Yaskawa INFORM job: kufsa_new.JBI

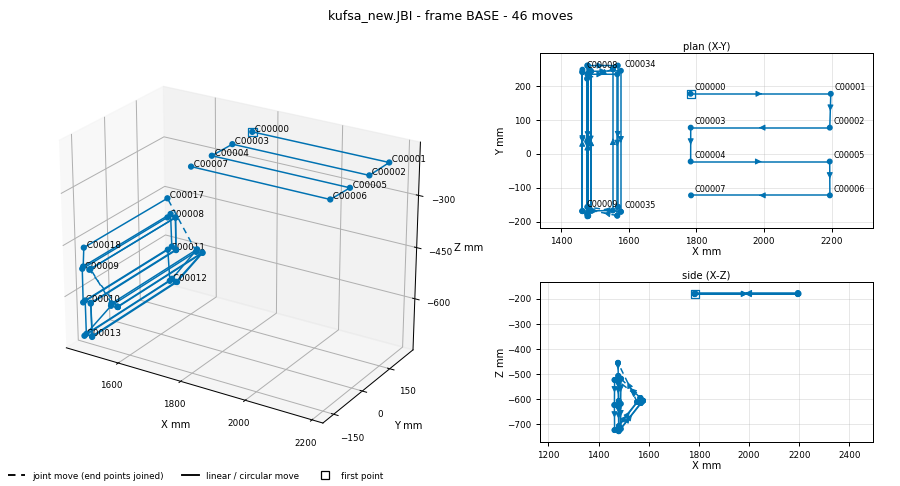
[picture p0: tool path of kufsa_new.JBI in frame BASE, 46 of 52 moves have a stored position in this frame; points joined in program order, loops and branches not executed]
/JOB
//NAME kufsa_new
//POS
///NPOS 46,0,46,0,0,0
///TOOL 0
///POSTYPE BASE
///RECTAN
///RCONF 1,0,0,0,0,0,0,0,0,0,0,0,0,0,0,0,0,0,0,0,0,0,0,0
C00000=1783.333,177.683,-178.952,175.0000,5.0000,90.0000
C00001=2197.437,177.683,-178.952,175.0000,5.0000,90.0000
C00002=2194.402,77.683,-180.929,175.0000,5.0000,90.0000
C00003=1783.689,77.683,-180.929,175.0000,5.0000,90.0000
C00004=1783.507,-22.316,-180.005,175.0000,5.0000,90.0000
C00005=2194.164,-22.316,-180.005,175.0000,5.0000,90.0000
C00006=2194.697,-122.316,-175.996,175.0000,5.0000,90.0000
C00007=1784.686,-122.316,-175.996,175.0000,5.0000,90.0000
C00008=1464.014,241.444,-522.722,175.0000,-89.9999,5.0000
C00009=1464.014,-169.159,-522.722,175.0000,-89.9999,5.0000
C00010=1463.152,-168.687,-622.722,175.0000,-89.9999,5.0000
C00011=1463.152,242.022,-622.722,175.0000,-89.9999,5.0000
C00012=1463.935,248.955,-722.722,175.0000,-89.9999,5.0000
C00013=1463.935,-168.695,-722.722,175.0000,-89.9999,5.0000
C00014=1553.861,-166.978,-610.590,180.0000,-45.0000,0.0000
C00015=1553.861,250.441,-610.590,180.0000,-45.0000,0.0000
C00016=1553.861,250.441,-610.590,180.0000,-45.0000,0.0000
C00017=1477.531,222.423,-454.518,175.0000,-89.9999,5.0000
C00018=1477.531,-177.571,-454.518,175.0000,-89.9999,5.0000
C00019=1478.554,-184.306,-506.723,175.0000,-89.9999,5.0000
C00020=1478.554,235.762,-506.723,175.0000,-89.9999,5.0000
C00021=1480.684,236.380,-606.723,175.0000,-89.9999,5.0000
C00022=1480.684,-183.074,-606.723,175.0000,-89.9999,5.0000
C00023=1480.955,-182.919,-706.723,175.0000,-89.9999,5.0000
C00024=1480.955,235.380,-706.723,175.0000,-89.9999,5.0000
C00025=1566.683,235.369,-594.591,180.0000,-45.0000,0.0000
C00026=1566.683,-182.153,-594.591,180.0000,-45.0000,0.0000
C00027=1566.683,-182.153,-594.591,180.0000,-45.0000,0.0000
C00028=1489.401,-166.687,-517.941,175.0000,-89.9999,5.0000
C00029=1489.401,243.705,-517.941,175.0000,-89.9999,5.0000
C00030=1488.117,245.937,-617.941,175.0000,-89.9999,5.0000
C00031=1488.117,-168.048,-617.941,175.0000,-89.9999,5.0000
C00032=1488.292,-166.510,-717.941,175.0000,-89.9999,5.0000
C00033=1488.292,243.987,-717.941,175.0000,-89.9999,5.0000
C00034=1577.392,245.653,-605.809,180.0000,-45.0000,0.0000
C00035=1577.392,-170.654,-605.809,180.0000,-45.0000,0.0000
C00036=1577.392,-170.654,-605.809,180.0000,-45.0000,0.0000
C00037=1478.179,-156.595,-527.111,175.0000,-89.9999,5.0000
C00038=1478.179,261.165,-527.111,175.0000,-89.9999,5.0000
C00039=1479.297,260.284,-627.111,175.0000,-89.9999,5.0000
C00040=1479.297,-156.550,-627.111,175.0000,-89.9999,5.0000
C00041=1480.372,-156.285,-727.111,175.0000,-89.9999,5.0000
C00042=1480.372,260.999,-727.111,175.0000,-89.9999,5.0000
C00043=1568.328,261.113,-614.979,180.0000,-45.0000,0.0000
C00044=1568.328,-156.025,-614.979,180.0000,-45.0000,0.0000
C00045=1568.328,-156.025,-614.979,180.0000,-45.0000,0.0000
///POSTYPE PULSE
///PULSE
EC00000=0
EC00001=0
EC00002=0
EC00003=0
EC00004=0
EC00005=0
EC00006=0
EC00007=0
EC00008=0
EC00009=0
EC00010=0
EC00011=0
EC00012=0
EC00013=0
EC00014=0
EC00015=0
EC00016=92160
EC00017=92160
EC00018=92160
EC00019=92160
EC00020=92160
EC00021=92160
EC00022=92160
EC00023=92160
EC00024=92160
EC00025=92160
EC00026=92160
EC00027=184320
EC00028=184320
EC00029=184320
EC00030=184320
EC00031=184320
EC00032=184320
EC00033=184320
EC00034=184320
EC00035=184320
EC00036=276480
EC00037=276480
EC00038=276480
EC00039=276480
EC00040=276480
EC00041=276480
EC00042=276480
EC00043=276480
EC00044=276480
EC00045=368640
//INST
///DATE 2023/01/19 11:30
///ATTR SC,RW,RJ
////FRAME BASE
///GROUP1 RB1,ST1
NOP
MOVJ P009 EX000 VJ=15.00
MOVJ C00000 EC00000 VJ=15.00
CALL JOB:SPYON
MOVL C00001 EC00001 V=200.0
MOVL C00002 EC00002 V=200.0
MOVL C00003 EC00003 V=200.0
MOVL C00004 EC00004 V=200.0
MOVL C00005 EC00005 V=200.0
MOVL C00006 EC00006 V=200.0
MOVL C00007 EC00007 V=200.0
CALL JOB:SPYOF
MOVJ P009 VJ=15.00
MOVJ C00008 EC00008 VJ=15.00
CALL JOB:SPYON
MOVL C00009 EC00009 V=200.0
MOVL C00010 EC00010 V=200.0
MOVL C00011 EC00011 V=200.0
MOVL C00012 EC00012 V=200.0
MOVL C00013 EC00013 V=200.0
MOVL C00014 EC00014 V=200.0
MOVL C00015 EC00015 V=200.0
CALL JOB:SPYOF
MOVJ P009 VJ=15.00
MOVL C00016 EC00016 V=200.0
MOVJ C00017 EC00017 VJ=15.00
CALL JOB:SPYON
MOVL C00018 EC00018 V=200.0
MOVL C00019 EC00019 V=200.0
MOVL C00020 EC00020 V=200.0
MOVL C00021 EC00021 V=200.0
MOVL C00022 EC00022 V=200.0
MOVL C00023 EC00023 V=200.0
MOVL C00024 EC00024 V=200.0
MOVL C00025 EC00025 V=200.0
MOVL C00026 EC00026 V=200.0
CALL JOB:SPYOF
MOVJ P009 VJ=15.00
MOVL C00027 EC00027 V=200.0
MOVJ C00028 EC00028 VJ=15.00
CALL JOB:SPYON
MOVL C00029 EC00029 V=200.0
MOVL C00030 EC00030 V=200.0
MOVL C00031 EC00031 V=200.0
MOVL C00032 EC00032 V=200.0
MOVL C00033 EC00033 V=200.0
MOVL C00034 EC00034 V=200.0
MOVL C00035 EC00035 V=200.0
CALL JOB:SPYOF
MOVJ P009 VJ=15.00
MOVL C00036 EC00036 V=200.0
MOVJ C00037 EC00037 VJ=15.00
CALL JOB:SPYON
MOVL C00038 EC00038 V=200.0
MOVL C00039 EC00039 V=200.0
MOVL C00040 EC00040 V=200.0
MOVL C00041 EC00041 V=200.0
MOVL C00042 EC00042 V=200.0
MOVL C00043 EC00043 V=200.0
MOVL C00044 EC00044 V=200.0
CALL JOB:SPYOF
MOVJ P009 VJ=15.00
MOVL C00045 EC00045 V=200.0
END
